ABB RobotStudio station: Task1+Task2.rspag

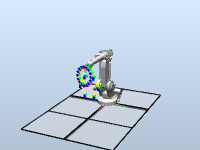
--- station ---
Station Solution2 (saved by RobotStudio 6.8.8148.134)
Controller System1
  mechanical unit ROB_1: IRB1410_5_144__01, 6 joints, base frame (0, 0, 0) mm
Layout (positions relative to the parent item):
  - IRB1410_5_144__01 [mechanism, from Robots\IRB1410_5_144_G_01.rslib] at (0, 0, 0) mm; joint values [0, 0, 0, 0, 0.5236, 0] (rad or m)
  - MyTool [mechanism, from Training Objects\myTool.rslib] at (943.61, 0, 1152.5) mm, rotated rx 180 ry 60 rz 180 deg
  - 部件_10 [part]
  - 部件_11 [part]
Attachment: MyTool is attached to IRB1410_5_144__01 / Link6

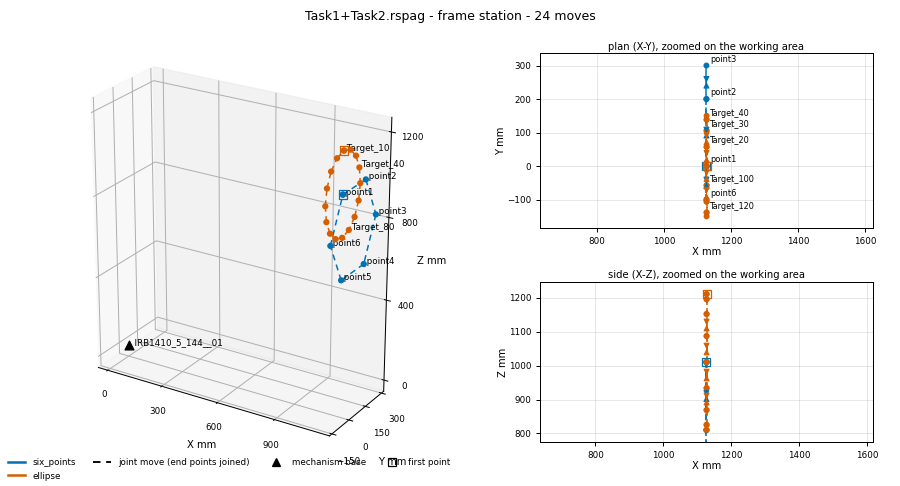
[picture p0: tool path of Task1+Task2.rspag in frame station, 24 of 24 moves have a stored position in this frame; points joined in program order, loops and branches not executed]
--- Backups/System1/RAPID/TASK1/PROGMOD/CalibData.mod ---
MODULE CalibData
	PERS tooldata MyTool:=[TRUE,[[31.7926,0,229.639],[0.945519,0,0.325568,0]],[1,[0,0,1],[1,0,0,0],0,0,0]];
ENDMODULE

--- Backups/System1/RAPID/TASK1/PROGMOD/Module1.mod ---
MODULE Module1
    CONST robtarget point1:=[[1126.588995348,0,1010.14730631],[0.190808996,0,0.981627183,0],[0,0,0,0],[9E+09,9E+09,9E+09,9E+09,9E+09,9E+09]];
    CONST robtarget point2:=[[1126.588995348,200,1010.14730631],[0.190808996,0,0.981627183,0],[0,0,0,0],[9E+09,9E+09,9E+09,9E+09,9E+09,9E+09]];
    CONST robtarget point3:=[[1126.588995348,300,810.14730631],[0.190808996,0,0.981627183,0],[0,-1,0,0],[9E+09,9E+09,9E+09,9E+09,9E+09,9E+09]];
    CONST robtarget point4:=[[1126.588995348,200,610.14730631],[0.017435796,-0.000761264,0.998896062,0.043612744],[0,0,-1,0],[9E+09,9E+09,9E+09,9E+09,9E+09,9E+09]];
    CONST robtarget point5:=[[1126.588995348,0,610.14730631],[0.190808996,0,0.981627183,0],[0,0,0,0],[9E+09,9E+09,9E+09,9E+09,9E+09,9E+09]];
    CONST robtarget point6:=[[1126.588995348,-100,810.14730631],[0.190808996,0,0.981627183,0],[0,0,0,0],[9E+09,9E+09,9E+09,9E+09,9E+09,9E+09]];

    CONST robtarget Target_10:=[[1127.053,0,1210.335],[0.704416026,0.061628417,0.704416026,0.061628417],[0,0,0,0],[9E+09,9E+09,9E+09,9E+09,9E+09,9E+09]];
    CONST robtarget Target_20:=[[1127.053,57.402514855,1195.110906502],[0.703798672,0.068318588,0.703798672,0.068318588],[0,0,-1,0],[9E+09,9E+09,9E+09,9E+09,9E+09,9E+09]];
    CONST robtarget Target_30:=[[1127.053,106.066017178,1151.756356237],[0.705836441,0.042366487,0.705836441,0.042366487],[0,0,-1,0],[9E+09,9E+09,9E+09,9E+09,9E+09,9E+09]];
    CONST robtarget Target_40:=[[1127.053,138.581929877,1086.871686473],[0.706904347,-0.016918744,0.706904347,-0.016918744],[0,0,-1,0],[9E+09,9E+09,9E+09,9E+09,9E+09,9E+09]];
    CONST robtarget Target_50:=[[1127.053,150,1010.335],[0.707106781,0,0.707106781,0],[0,0,-1,0],[9E+09,9E+09,9E+09,9E+09,9E+09,9E+09]];
    CONST robtarget Target_60:=[[1127.053,138.581929877,933.798313527],[0.706904347,0.016918744,0.706904347,0.016918744],[0,-1,-1,0],[9E+09,9E+09,9E+09,9E+09,9E+09,9E+09]];
    CONST robtarget Target_70:=[[1127.053,106.066017178,868.913643763],[0.742463059,0.067513368,0.665843444,-0.029035488],[0,-1,-1,0],[9E+09,9E+09,9E+09,9E+09,9E+09,9E+09]];
    CONST robtarget Target_80:=[[1127.053,57.402514855,825.559093498],[0.707074863,-0.006718519,0.707074863,-0.006718519],[-1,-1,-1,0],[9E+09,9E+09,9E+09,9E+09,9E+09,9E+09]];
    CONST robtarget Target_90:=[[1127.053,0,810.335],[0.707106781,0,0.707106781,0],[-1,-1,-1,0],[9E+09,9E+09,9E+09,9E+09,9E+09,9E+09]];
    CONST robtarget Target_100:=[[1127.053,-57.402514855,825.559093498],[0.766009868,0.007278516,0.64275859,0.006107398],[-1,-1,0,0],[9E+09,9E+09,9E+09,9E+09,9E+09,9E+09]];
    CONST robtarget Target_110:=[[1127.053,-106.066017178,868.913643763],[0.706843002,-0.01931243,0.706843002,-0.01931243],[-1,-1,0,0],[9E+09,9E+09,9E+09,9E+09,9E+09,9E+09]];
    CONST robtarget Target_120:=[[1127.053,-138.581929877,933.798313527],[0.699102791,0.106090941,0.699102791,0.106090941],[-1,0,0,0],[9E+09,9E+09,9E+09,9E+09,9E+09,9E+09]];
    CONST robtarget Target_130:=[[1127.053,-150,1010.335],[0.707106781,0,0.707106781,0],[-1,-1,0,0],[9E+09,9E+09,9E+09,9E+09,9E+09,9E+09]];
    CONST robtarget Target_140:=[[1127.053,-138.581929877,1086.871686473],[0.706904347,0.016918744,0.706904347,0.016918744],[-1,-1,0,0],[9E+09,9E+09,9E+09,9E+09,9E+09,9E+09]];
    CONST robtarget Target_150:=[[1127.053,-106.066017178,1151.756356237],[0.706843002,0.019312429,0.706843002,0.019312429],[0,0,0,0],[9E+09,9E+09,9E+09,9E+09,9E+09,9E+09]];
    CONST robtarget Target_160:=[[1127.053,-57.402514855,1195.110906502],[0.704969787,0.054932681,0.704969787,0.054932681],[0,0,0,0],[9E+09,9E+09,9E+09,9E+09,9E+09,9E+09]];
    CONST robtarget Target_170:=[[1127.053,0,1210.335],[0.707106781,0,0.707106781,0],[0,0,0,0],[9E+09,9E+09,9E+09,9E+09,9E+09,9E+09]];
    CONST robtarget point7:=[[1368.131468028,17.364817855,1111.854224714],[0.704416026,0.061628417,0.704416026,0.061628417],[0,0,0,0],[9E+09,9E+09,9E+09,9E+09,9E+09,9E+09]];


    PROC main()
        six_points;
        ellipse;

    ENDPROC
    PROC six_points()
        MoveJ point1,v100,z10,MyTool\WObj:=wobj0;
        MoveJ point2,v100,z10,MyTool\WObj:=wobj0;
        MoveJ point3,v100,z10,MyTool\WObj:=wobj0;
        MoveJ point4,v100,z10,MyTool\WObj:=wobj0;
        MoveJ point5,v100,z10,MyTool\WObj:=wobj0;
        MoveJ point6,v100,z10,MyTool\WObj:=wobj0;
        MoveJ point1,v100,z10,MyTool\WObj:=wobj0;
    ENDPROC

	PROC ellipse()
	    MoveJ Target_10,v100,z10,MyTool\WObj:=wobj0;
	    MoveJ Target_20,v100,z10,MyTool\WObj:=wobj0;
	    MoveJ Target_30,v100,z10,MyTool\WObj:=wobj0;
	    MoveJ Target_40,v100,z10,MyTool\WObj:=wobj0;
	    MoveJ Target_50,v100,z10,MyTool\WObj:=wobj0;
	    MoveJ Target_60,v100,z10,MyTool\WObj:=wobj0;
	    MoveJ Target_70,v100,z10,MyTool\WObj:=wobj0;
	    MoveJ Target_80,v100,z10,MyTool\WObj:=wobj0;
	    MoveJ Target_90,v100,z10,MyTool\WObj:=wobj0;
	    MoveJ Target_100,v100,z10,MyTool\WObj:=wobj0;
	    MoveJ Target_110,v100,z10,MyTool\WObj:=wobj0;
	    MoveJ Target_120,v100,z10,MyTool\WObj:=wobj0;
	    MoveJ Target_130,v100,z10,MyTool\WObj:=wobj0;
	    MoveJ Target_140,v100,z10,MyTool\WObj:=wobj0;
	    MoveJ Target_150,v100,z10,MyTool\WObj:=wobj0;
	    MoveJ Target_160,v100,z10,MyTool\WObj:=wobj0;
	    MoveJ Target_170,v100,z10,MyTool\WObj:=wobj0;
	ENDPROC


ENDMODULE
